TYPE typeStationComplexity :
STRUCT
	task:UINT;
	complexity:uint;
	
END_STRUCT
END_TYPE

(* stored: Version 1.1.0.1, ProductVersion 3.1.4024.12
   DUT typeStationComplexity: Id {975719f8-dc18-43c6-b636-e6b8da523bb0} *)
